// TIA Portal project "2022.11.02—跑马灯" (V17)

(* hardware
DEVICE "S7-1200 station_1"  S7-1200 Station
   slot 0: "Rack_0"  S7-1200 Rack  Rack  V1.0
   slot 1: "PLC_1"  CPU 1214C DC/DC/Rly  6ES7 214-1HG40-0XB0  V4.5
DEVICE "HMI_1"  KTP700 Basic PN
   slot 0: "HMI_1"  KTP700 Basic PN  6AV2 123-2GB03-0AX0  17.0.0.0
   slot 1: "HMI_RT_1"  KTP700 Basic PN  6AV2 123-2GB03-0AX0  17.0.0.0
   slot 5: "HMI_1.IE_CP_1"  PROFINET Interface  17.0.0.0
      slot 1: "PROFINET Interface_1"  PROFINET Interface
         slot 1: "Port_1"  Port
*)

// ===== PLC "PLC_1"  CPU 1214C DC/DC/Rly =====

VAR_GLOBAL   // PLC tag table "默认变量表"
   "源操作数1" AT %MW6 : Word;
   "目标操作数1" AT %MW10 : Word;
   "源操作数2" AT %MD20 : DWord;
   "目标操作数2" AT %MD100 : DWord;
   "运行标志位" AT %M4.0 : Bool;
   "启动" AT %M3.0 : Bool;
   "停止" AT %M3.1 : Bool;
   "当前值" AT %MD6 : Time;
   "LED灯带" AT %MW16 : Int;
END_VAR

VAR_GLOBAL   // PLC tag table "LED"
   "1LED_1" AT %M16.0 : Bool;
   "1LED_2" AT %M16.1 : Bool;
   "1LED_3" AT %M16.2 : Bool;
   "1LED_4" AT %M16.3 : Bool;
   "2LED_1" AT %M16.4 : Bool;
   "2LED_2" AT %M16.5 : Bool;
   "2LED_3" AT %M16.6 : Bool;
   "2LED_4" AT %M16.7 : Bool;
   "3LED_1" AT %M17.0 : Bool;
   "3LED_2" AT %M17.1 : Bool;
   "3LED_3" AT %M17.2 : Bool;
   "3LED_4" AT %M17.3 : Bool;
   "4LED_1" AT %M17.4 : Bool;
   "4LED_2" AT %M17.5 : Bool;
   "4LED_3" AT %M17.6 : Bool;
   "4LED_4" AT %M17.7 : Bool;
END_VAR

DATA_BLOCK "数据块_1"   // DB1
{ S7_Optimized_Access := 'TRUE' }
VERSION : 0.1
   VAR
      "a" : DWord;
      "b" : DWord;
   END_VAR
BEGIN
END_DATA_BLOCK

DATA_BLOCK "数据块_2"   // DB2
{ S7_Optimized_Access := 'TRUE' }
VERSION : 0.1
   VAR
      c : DInt;
   END_VAR
BEGIN
END_DATA_BLOCK

// folder: System blocks/Program resources

DATA_BLOCK "IEC_Timer_0_DB"   // DB3
{ S7_Optimized_Access := 'TRUE' }
AUTHOR : Simatic
FAMILY : IEC
NAME : IEC_TMR
VERSION : 1.0
// stored: InstanceOfName IEC_TIMER
"IEC_TIMER"
BEGIN
END_DATA_BLOCK

// folder: (top level)

ORGANIZATION_BLOCK "Main"   // OB1, LAD, ProgramCycle
TITLE = "Main Program Sweep (Cycle)"
{ S7_Optimized_Access := 'TRUE' }
VERSION : 0.1
   VAR_INPUT
      Initial_Call : Bool;   // Initial call of this OB
      Remanence : Bool;   // =True, if remanent data are available
   END_VAR
BEGIN

REGION Network 1: 移动指令
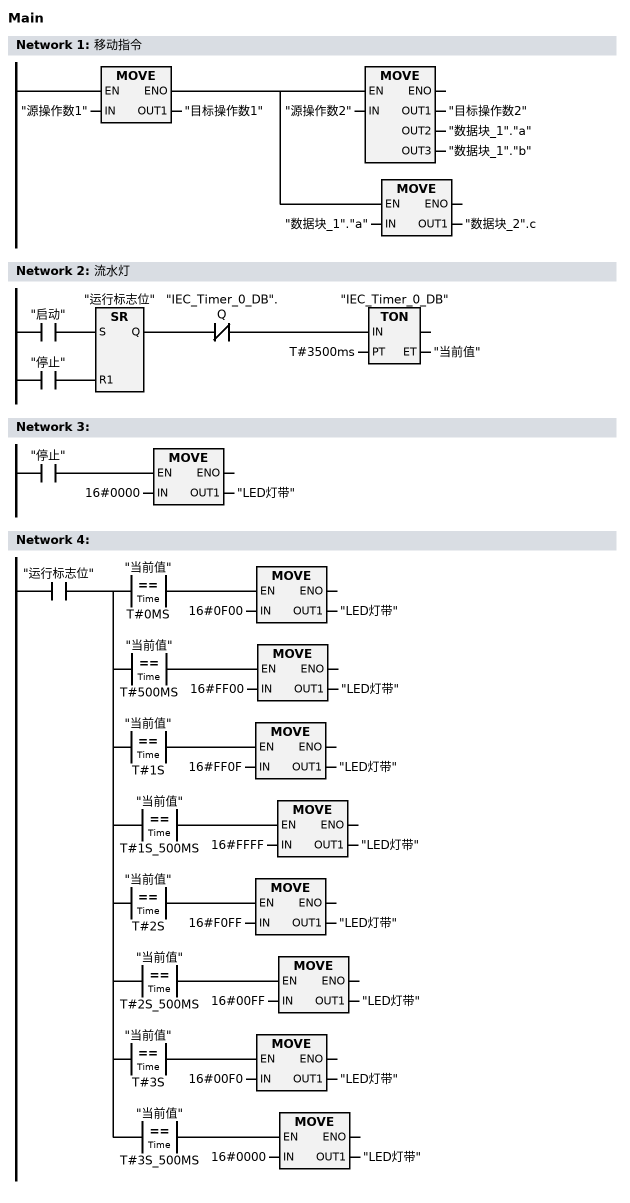
   RUNG wire#powerrail
      Move(in := "源操作数1", out1 => "目标操作数1")
      wire#w1
      Move(in := "源操作数2", out1 => "目标操作数2", out2 => "数据块_1"."a", out3 => "数据块_1"."b")
   END_RUNG
   RUNG wire#w1
      Move(in := "数据块_1"."a", out1 => "数据块_2".c)
   END_RUNG
   // the same network as SCL:
   "目标操作数1" := "源操作数1";
   "目标操作数2" := "源操作数2";
   "数据块_1"."a" := "源操作数2";
   "数据块_1"."b" := "源操作数2";
   "数据块_2".c := "数据块_1"."a";
END_REGION

REGION Network 2: 流水灯
   IF "启动" THEN
       "运行标志位" := TRUE;   // SR flip-flop
   END_IF;
   IF "停止" THEN "运行标志位" := FALSE; END_IF;
   "IEC_Timer_0_DB".TON(IN := "运行标志位" AND NOT "IEC_Timer_0_DB".Q, PT := T#3500ms, ET => "当前值");
END_REGION

REGION Network 3
   RUNG wire#powerrail
      Contact( "停止" )
      Move(in := 16#0000, out1 => "LED灯带")
   END_RUNG
   // the same network as SCL:
   IF "停止" THEN "LED灯带" := 16#0000; END_IF;
END_REGION

REGION Network 4
   RUNG wire#powerrail
      Contact( "运行标志位" )
      wire#w1
      { S7_Templates := "SrcType := Time" } EQ_Contact(in1 := "当前值", in2 := T#0MS)
      Move(in := 16#0F00, out1 => "LED灯带")
   END_RUNG
   RUNG wire#w1
      { S7_Templates := "SrcType := Time" } EQ_Contact(in1 := "当前值", in2 := T#500MS)
      Move(in := 16#FF00, out1 => "LED灯带")
   END_RUNG
   RUNG wire#w1
      { S7_Templates := "SrcType := Time" } EQ_Contact(in1 := "当前值", in2 := T#1S)
      Move(in := 16#FF0F, out1 => "LED灯带")
   END_RUNG
   RUNG wire#w1
      { S7_Templates := "SrcType := Time" } EQ_Contact(in1 := "当前值", in2 := T#1S_500MS)
      Move(in := 16#FFFF, out1 => "LED灯带")
   END_RUNG
   RUNG wire#w1
      { S7_Templates := "SrcType := Time" } EQ_Contact(in1 := "当前值", in2 := T#2S)
      Move(in := 16#F0FF, out1 => "LED灯带")
   END_RUNG
   RUNG wire#w1
      { S7_Templates := "SrcType := Time" } EQ_Contact(in1 := "当前值", in2 := T#2S_500MS)
      Move(in := 16#00FF, out1 => "LED灯带")
   END_RUNG
   RUNG wire#w1
      { S7_Templates := "SrcType := Time" } EQ_Contact(in1 := "当前值", in2 := T#3S)
      Move(in := 16#00F0, out1 => "LED灯带")
   END_RUNG
   RUNG wire#w1
      { S7_Templates := "SrcType := Time" } EQ_Contact(in1 := "当前值", in2 := T#3S_500MS)
      Move(in := 16#0000, out1 => "LED灯带")
   END_RUNG
   // the same network as SCL:
   IF "运行标志位" AND ("当前值" = T#0MS) THEN "LED灯带" := 16#0F00; END_IF;
   IF "运行标志位" AND ("当前值" = T#500MS) THEN "LED灯带" := 16#FF00; END_IF;
   IF "运行标志位" AND ("当前值" = T#1S) THEN "LED灯带" := 16#FF0F; END_IF;
   IF "运行标志位" AND ("当前值" = T#1S_500MS) THEN "LED灯带" := 16#FFFF; END_IF;
   IF "运行标志位" AND ("当前值" = T#2S) THEN "LED灯带" := 16#F0FF; END_IF;
   IF "运行标志位" AND ("当前值" = T#2S_500MS) THEN "LED灯带" := 16#00FF; END_IF;
   IF "运行标志位" AND ("当前值" = T#3S) THEN "LED灯带" := 16#00F0; END_IF;
   IF "运行标志位" AND ("当前值" = T#3S_500MS) THEN "LED灯带" := 16#0000; END_IF;
END_REGION
END_ORGANIZATION_BLOCK

(* ===== HMI "HMI_RT_1" =====
system functions are stored by id; their names below are inferred from use
connection "HMI_连接_1": ETHERNET, SMART_S7_1200_OMS

HMI tags "默认变量表"
   "Tag_ScreenNumber" : UInt, internal
   "1LED_1" : Bool = PLC 1LED_1 AT %M16.0, 1 s
   "1LED_2" : Bool = PLC 1LED_2 AT %M16.1, 1 s
   "2LED_1" : Bool = PLC 2LED_1 AT %M16.4, 1 s
   "3LED_1" : Bool = PLC 3LED_1 AT %M17.0, 1 s
   "4LED_1" : Bool = PLC 4LED_1 AT %M17.4, 1 s
   "启动" : Bool = PLC 启动 AT %M3.0, 1 s
   "停止" : Bool = PLC 停止 AT %M3.1, 1 s

Template "模板_1" 800x480
   Button "退出" at 714,429 size 71x50; TextOff '退出'; PictureOff "ExitRuntime_KTP700_Basic_PN_TR"; PictureOn "ExitRuntime_KTP700_Basic_PN_TR"
      on Release: StopRuntime(0)
   Button "Template_Button" at 614,429 size 71x50; TextOff 'Text'
   Button "Template_Button_1" at 514,429 size 71x50; TextOff 'Text'
   Button "Template_Button_2" at 414,429 size 71x50; TextOff 'Text'
   Button "Template_Button_3" at 314,429 size 71x50; TextOff 'Text'
   Button "Template_Button_4" at 214,429 size 71x50; TextOff 'Text'
   Button "报警" at 114,429 size 71x50; TextOff '报警'; PictureOff "AlarmDisplay_KTP700_Basic_PN_TR"; PictureOn "AlarmDisplay_KTP700_Basic_PN_TR"
      on Release: function_ef3f5d25("报警窗口_Unacknowledged", -1)
   Button "起始画面" at 14,429 size 71x50; TextOff '起始画面'; PictureOff "NavigateHome_KTP700_Basic_PN_TR"; PictureOn "NavigateHome_KTP700_Basic_PN_TR"
      on Release: ActivateScreen("根画面", 0)
   SymbolicIOField "Symbolic_IO_Field_Screen" at 93,9 size 600x33; TextOff '0'; TextOn '1'; TextList "TextList_ScreenNames"
      ProcessValue <- "Tag_ScreenNumber"
      on Change: ActivateScreenByNumber("Tag_ScreenNumber", 0)
   DateTimeField "HmiScreenItemData" at 695,25 size 105x25
   DateTimeField "HmiScreenItemData_1" at 695,0 size 105x25
   GraphicView "Logo" at 0,0 size 91x51; Picture "HMI_1 的 Logo"

screen "根画面" 800x480, template "模板_1"
   on GenerateScreen: SetTag("Tag_ScreenNumber", 1)
   Rectangle "矩形_1" at 304,164 size 118x11
      Appearance <- "1LED_1"
   Rectangle "矩形_2" at 242,108 size 250x11
      Appearance <- "3LED_1"
   Rectangle "矩形_3" at 278,139 size 174x11
      Appearance <- "2LED_1"
   Rectangle "矩形_6" at 420,175 size 12x93
      Appearance <- "1LED_2"
   Rectangle "矩形_16" at 209,67 size 321x11
      Appearance <- "4LED_1"
   Button "按钮_1" at 600,153 size 96x32; TextOff '启动'
      on Press: SetBit("启动")
      on Release: ResetBit("启动")
   Button "按钮_2" at 600,205 size 96x32; TextOff '停止'
      on Press: SetBit("停止")
      on Release: ResetBit("停止")
*)